(* Schneider Machine Expert - Basic project task1trial3, file version 2.7.0.0 *)
(* ProjectInformations: Name=New project *)

HARDWARE
  Cpu 0: TM221CE40T
  EthernetConfiguration: NetworkName=M221, IpAllocationMode=FixedAddress, IpAddress=0.0.0.0, SubnetMask=0.0.0.0
  SerialLineConfiguration: Baud=Baud19200, Parity=ParityEven, DataBits=DataBits8, StopBits=StopBits1, PhysicalMedium=PhysicalMediumRs485, TransmissionMode=TransmissionModeModbusRtu, SlaveId=1, Addressing=SlaveAddressing
  MastTask: UsePeriodScanMode=false, PeriodScan=100
  FastTask: Period=255
  CpuBehavior: StartingMode=StartAsPreviousState, AutoSaveRamOnEeprom=true, WatchdogPeriod=250

SYMBOLS  (address, symbol, comment, settings)
  %M0       POWERMEMORY
  %M1       SENSOR1MEMORY
  %M2       SENSOR2MEMORY
  %TM0        [Preset=5, Base=OneSecond]
  %I0.0     START_BUTTON
  %I0.1     EMERGENCY
  %I0.2     SENSORSTART
  %I0.3     SENSORSTOP
  %Q0.0     POWER
  %Q0.1     LAMPU
  %Q0.2     MOTOR
  %Q0.3     TIMERSENSOR

POU New POU
  (* SectionNumber=1 *)

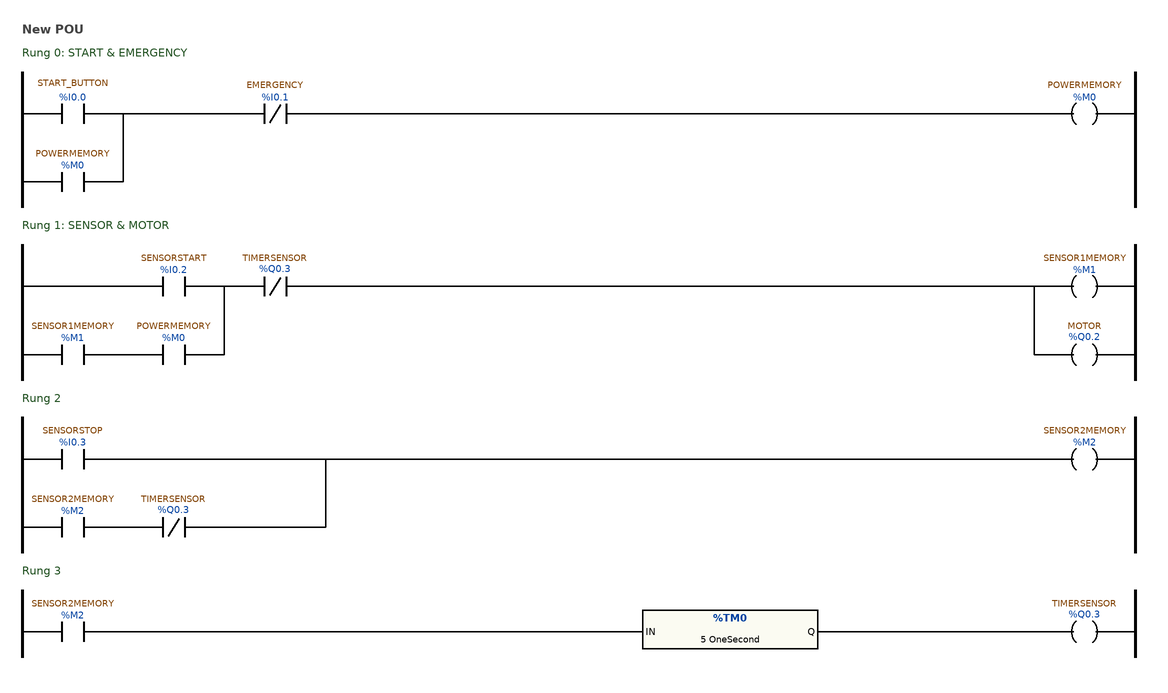

// Rung 0: START & EMERGENCY
  LD %I0.0                (* START_BUTTON *)
  OR %M0                  (* POWERMEMORY *)
  ANDN %I0.1              (* EMERGENCY *)
  ST %M0                  (* POWERMEMORY *)
  // as ST:
  //   POWERMEMORY := (START_BUTTON OR POWERMEMORY) AND NOT EMERGENCY;

// Rung 1: SENSOR & MOTOR
  LD %I0.2                (* SENSORSTART *)
  OR( %M1                 (* SENSOR1MEMORY *)
  AND %M0                 (* POWERMEMORY *)
  )
  ANDN %Q0.3              (* TIMERSENSOR *)
  ST %M1                  (* SENSOR1MEMORY *)
  ST %Q0.2                (* MOTOR *)
  // as ST:
  //   _t1 := (SENSORSTART OR SENSOR1MEMORY AND POWERMEMORY) AND NOT TIMERSENSOR;
  //   SENSOR1MEMORY := _t1;
  //   MOTOR := _t1;

// Rung 2
  LD %I0.3                (* SENSORSTOP *)
  OR( %M2                 (* SENSOR2MEMORY *)
  ANDN %Q0.3              (* TIMERSENSOR *)
  )
  ST %M2                  (* SENSOR2MEMORY *)
  // as ST:
  //   SENSOR2MEMORY := SENSORSTOP OR SENSOR2MEMORY AND NOT TIMERSENSOR;

// Rung 3
  BLK %TM0
  LD %M2                  (* SENSOR2MEMORY *)
  IN
  OUT_BLK
  LD Q
  ST %Q0.3                (* TIMERSENSOR *)
  END_BLK
  // as ST:
  //   %TM0(IN := SENSOR2MEMORY);
  //   TIMERSENSOR := %TM0.Q;
